// TIA Portal project "time_series_GV" (V14)

(* hardware
DEVICE "S71500/ET200MP station_1"  S7-1500 station
   slot 0: "Rail_0"  Rack  6ES7 590-1***0-0AA0
   slot 0: "PM 70W 120/230VAC"  PM 70W 120/230VAC  6EP1332-4BA00
   slot 1: "PLC_1"  CPU 1511-1 PN  6ES7 511-1AK01-0AB0  V2.1
      slot 3: "CPU display_1"  6ES7591-1AA00-0AA0
   slot 2: "DI 16/DQ 16x24VDC/0.5A BA_1"  DI 16/DQ 16x24VDC/0.5A BA  6ES7 523-1BL00-0AA0  V1.0
   slot 3: "AI/AQ 4xU/I/RTD/TC / 2xU/I ST_1"  AI/AQ 4xU/I/RTD/TC / 2xU/I ST  6ES7 534-7QE00-0AB0  V1.0
DEVICE "HMI_1"  KTP900 Basic PN
   slot 0: "KTP900 Basic PN"  KTP900 Basic PN  6AV2 123-2JB03-0AX0  14.0.1.0
   slot 1: "HMI_RT_1"  KTP900 Basic PN  6AV2 123-2JB03-0AX0  14.0.1.0
   slot 5: "HMI_1.IE_CP_1"  PROFINET Interface  14.0.1.0
      slot 1: "PROFINET Interface_1"  PROFINET Interface
         slot 1: "Port_1"  Port
*)

// ===== PLC "PLC_1"  CPU 1511-1 PN =====

VAR_GLOBAL   // PLC tag table "Default tag table"
   "System_Byte" AT %MB1 : Byte;
   "FirstScan" AT %M1.0 : Bool;
   "DiagStatusUpdate" AT %M1.1 : Bool;
   "AlwaysTRUE" AT %M1.2 : Bool;
   "AlwaysFALSE" AT %M1.3 : Bool;
   "Clock_Byte" AT %MB0 : Byte;
   "Clock_10Hz" AT %M0.0 : Bool;
   "Clock_5Hz" AT %M0.1 : Bool;
   "Clock_2.5Hz" AT %M0.2 : Bool;
   "Clock_2Hz" AT %M0.3 : Bool;
   "Clock_1.25Hz" AT %M0.4 : Bool;
   "Clock_1Hz" AT %M0.5 : Bool;
   "Clock_0.625Hz" AT %M0.6 : Bool;
   "Clock_0.5Hz" AT %M0.7 : Bool;
   "Out_Standart_Deviation" AT %MD2 : Real;
   "Cloc_frequence" AT %M6.0 : Bool;
   "countdown_Frequency" AT %MD8 : Time;
   "arithmetic_avg" AT %MD12 : Real;
   "stdt_out" AT %MD16 : Real;
   "error_avg" AT %M6.1 : Bool;
   "status_id" AT %MW20 : UInt;
   "status_bloc" AT %MW22 : Word;
   "ret_val_DB" AT %MW28 : Int;
   "value_read_array" AT %MW24 : Int;
   "ret_val_DB_read" AT %MW26 : Int;
   "size_array_block" AT %MW30 : Int;
   "signal_out_analog" AT %MW32 : Int;
   "standartDeviation" AT %MD34 : Real;
END_VAR

DATA_BLOCK "DB_Signal_measurement"   // DB1
{ S7_Optimized_Access := 'TRUE' }
VERSION : 0.1
   VAR
      Signal : Array[0..15] of Int;
   END_VAR
BEGIN
   Signal[0] := 1;
   Signal[1] := 2;
   Signal[2] := 3;
   Signal[4] := 5;
   Signal[3] := 4;
   Signal[5] := 6;
   Signal[6] := 7;
   Signal[7] := 8;
   Signal[8] := 9;
   Signal[9] := 0;
   Signal[10] := 1;
   Signal[11] := 2;
   Signal[12] := 3;
   Signal[13] := 4;
   Signal[14] := 5;
   Signal[15] := 6;
END_DATA_BLOCK

DATA_BLOCK "Array_DB_Signal"   // DB2
{ S7_Optimized_Access := 'TRUE' }
VERSION : 0.1
   VAR
      Header : ArrayDBHeader;
      THIS : Array[0..15] of Real;
   END_VAR
BEGIN
   Header.LowerBound := 0;
   Header.UpperBound := 15;
   Header.Elements := 16;
   Header.PaddedSize := 4;
   Header.ElementSize := 4;
   THIS[0] := 8.0;
   THIS[1] := 6.2;
   THIS[2] := 7.5;
   THIS[3] := 8.5;
   THIS[4] := 7.0;
   THIS[5] := 2.8;
   THIS[8] := 100.0;
   THIS[9] := 100.0;
END_DATA_BLOCK

DATA_BLOCK "HMI_Signal"   // DB3
{ S7_Optimized_Access := 'TRUE' }
VERSION : 0.1
   VAR
      HMI_signal_out_GV : Int;
      HMI_stdDeviation : Real;
   END_VAR
BEGIN
END_DATA_BLOCK

DATA_BLOCK "myArrayDB"   // DB4
{ S7_Optimized_Access := 'TRUE' }
VERSION : 0.1
   VAR
      Header : ArrayDBHeader;
      THIS : Array[0..1300] of Int;
   END_VAR
BEGIN
   Header.LowerBound := 0;
   Header.UpperBound := 1300;
   Header.Elements := 1301;
   Header.PaddedSize := 2;
   Header.ElementSize := 2;
   THIS[4] := 659;
   THIS[0] := 620;
   THIS[1] := 620;
   THIS[2] := 620;
   THIS[3] := 650;
   THIS[5] := 659;
   THIS[6] := 659;
   THIS[7] := 676;
   THIS[8] := 676;
   THIS[9] := 676;
   THIS[10] := 676;
   THIS[11] := 676;
   THIS[12] := 676;
   THIS[13] := 676;
   THIS[14] := 677;
   THIS[15] := 677;
   THIS[16] := 677;
   THIS[17] := 677;
   THIS[18] := 677;
   THIS[19] := 677;
   THIS[20] := 677;
   THIS[21] := 677;
   THIS[22] := 677;
   THIS[23] := 677;
   THIS[24] := 677;
   THIS[25] := 678;
   THIS[26] := 678;
   THIS[27] := 678;
   THIS[28] := 678;
   THIS[29] := 678;
   THIS[30] := 678;
   THIS[31] := 678;
   THIS[32] := 678;
   THIS[33] := 678;
   THIS[34] := 678;
   THIS[35] := 678;
   THIS[36] := 678;
   THIS[37] := 678;
   THIS[38] := 678;
   THIS[39] := 678;
   THIS[40] := 678;
   THIS[41] := 678;
   THIS[42] := 672;
   THIS[43] := 663;
   THIS[44] := 663;
   THIS[45] := 663;
   THIS[46] := 630;
   THIS[47] := 627;
   THIS[48] := 627;
   THIS[49] := 617;
   THIS[50] := 617;
   THIS[51] := 617;
   THIS[52] := 617;
   THIS[53] := 617;
   THIS[54] := 617;
   THIS[55] := 617;
   THIS[56] := 618;
   THIS[57] := 620;
   THIS[58] := 620;
   THIS[59] := 620;
   THIS[60] := 621;
   THIS[61] := 621;
   THIS[62] := 621;
   THIS[63] := 621;
   THIS[64] := 621;
   THIS[65] := 621;
   THIS[66] := 621;
   THIS[67] := 621;
   THIS[68] := 621;
   THIS[69] := 621;
   THIS[70] := 621;
   THIS[71] := 621;
   THIS[72] := 621;
   THIS[73] := 621;
   THIS[74] := 621;
   THIS[75] := 621;
   THIS[76] := 621;
   THIS[77] := 621;
   THIS[78] := 621;
   THIS[79] := 621;
   THIS[80] := 621;
   THIS[81] := 618;
   THIS[82] := 612;
   THIS[83] := 612;
   THIS[84] := 595;
   THIS[85] := 584;
   THIS[86] := 584;
   THIS[87] := 579;
   THIS[88] := 579;
   THIS[89] := 579;
   THIS[90] := 579;
   THIS[91] := 579;
   THIS[92] := 579;
   THIS[93] := 579;
   THIS[94] := 579;
   THIS[95] := 579;
   THIS[96] := 579;
   THIS[97] := 579;
   THIS[98] := 579;
   THIS[99] := 579;
   THIS[100] := 579;
   THIS[101] := 579;
   THIS[102] := 579;
   THIS[103] := 579;
   THIS[104] := 579;
   THIS[105] := 579;
   THIS[106] := 579;
   THIS[107] := 579;
   THIS[108] := 579;
   THIS[109] := 579;
   THIS[110] := 579;
   THIS[111] := 579;
   THIS[112] := 579;
   THIS[113] := 579;
   THIS[114] := 579;
   THIS[115] := 579;
   THIS[116] := 579;
   THIS[117] := 579;
   THIS[118] := 579;
   THIS[119] := 579;
   THIS[120] := 579;
   THIS[121] := 579;
   THIS[122] := 579;
   THIS[123] := 572;
   THIS[124] := 564;
   THIS[125] := 564;
   THIS[126] := 551;
   THIS[127] := 548;
   THIS[128] := 548;
   THIS[129] := 548;
   THIS[130] := 545;
   THIS[131] := 545;
   THIS[132] := 541;
   THIS[133] := 541;
   THIS[134] := 541;
   THIS[135] := 541;
   THIS[136] := 541;
   THIS[137] := 542;
   THIS[138] := 542;
   THIS[139] := 542;
   THIS[140] := 542;
   THIS[141] := 542;
   THIS[142] := 542;
   THIS[143] := 542;
   THIS[144] := 542;
   THIS[145] := 542;
   THIS[146] := 542;
   THIS[147] := 542;
   THIS[148] := 542;
   THIS[149] := 542;
   THIS[150] := 538;
   THIS[151] := 532;
   THIS[152] := 532;
   THIS[153] := 518;
   THIS[154] := 511;
   THIS[155] := 511;
   THIS[156] := 511;
   THIS[157] := 508;
   THIS[158] := 508;
   THIS[159] := 508;
   THIS[160] := 508;
   THIS[161] := 508;
   THIS[162] := 508;
   THIS[163] := 508;
   THIS[164] := 508;
   THIS[165] := 508;
   THIS[166] := 508;
   THIS[167] := 508;
   THIS[168] := 508;
   THIS[169] := 501;
   THIS[170] := 500;
   THIS[171] := 500;
   THIS[172] := 500;
   THIS[173] := 500;
   THIS[174] := 500;
   THIS[175] := 500;
   THIS[176] := 500;
   THIS[177] := 500;
   THIS[178] := 520;
   THIS[179] := 521;
   THIS[180] := 521;
   THIS[181] := 420;
   THIS[182] := 500;
   THIS[183] := 500;
   THIS[184] := 500;
   THIS[185] := 500;
   THIS[186] := 500;
   THIS[187] := 500;
   THIS[188] := 500;
   THIS[189] := 500;
   THIS[190] := 481;
   THIS[191] := 481;
   THIS[192] := 481;
   THIS[193] := 463;
   THIS[194] := 463;
   THIS[195] := 463;
   THIS[196] := 461;
   THIS[197] := 461;
   THIS[198] := 461;
   THIS[199] := 461;
   THIS[200] := 461;
   THIS[201] := 461;
   THIS[202] := 461;
   THIS[203] := 461;
   THIS[204] := 461;
   THIS[205] := 461;
   THIS[206] := 461;
   THIS[207] := 461;
   THIS[208] := 461;
   THIS[209] := 461;
   THIS[210] := 461;
   THIS[211] := 461;
   THIS[212] := 459;
   THIS[213] := 458;
   THIS[214] := 447;
   THIS[215] := 441;
   THIS[216] := 434;
   THIS[217] := 427;
   THIS[218] := 426;
   THIS[219] := 426;
   THIS[220] := 426;
   THIS[221] := 426;
   THIS[222] := 426;
   THIS[223] := 426;
   THIS[224] := 426;
   THIS[225] := 426;
   THIS[226] := 426;
   THIS[227] := 426;
   THIS[228] := 426;
   THIS[229] := 426;
   THIS[230] := 426;
   THIS[231] := 426;
   THIS[232] := 426;
   THIS[233] := 426;
   THIS[234] := 426;
   THIS[235] := 426;
   THIS[236] := 426;
   THIS[237] := 426;
   THIS[238] := 426;
   THIS[239] := 426;
   THIS[240] := 426;
   THIS[241] := 426;
   THIS[242] := 426;
   THIS[243] := 426;
   THIS[244] := 426;
   THIS[245] := 426;
   THIS[246] := 426;
   THIS[247] := 426;
   THIS[248] := 426;
   THIS[249] := 426;
   THIS[250] := 426;
   THIS[251] := 426;
   THIS[252] := 426;
   THIS[253] := 426;
   THIS[254] := 426;
   THIS[255] := 426;
   THIS[256] := 426;
   THIS[257] := 426;
   THIS[258] := 421;
   THIS[259] := 415;
   THIS[260] := 415;
   THIS[261] := 401;
   THIS[262] := 398;
   THIS[263] := 392;
   THIS[264] := 392;
   THIS[265] := 389;
   THIS[266] := 389;
   THIS[267] := 389;
   THIS[268] := 389;
   THIS[269] := 385;
   THIS[270] := 384;
   THIS[271] := 384;
   THIS[272] := 384;
   THIS[273] := 384;
   THIS[274] := 384;
   THIS[275] := 384;
   THIS[276] := 384;
   THIS[277] := 384;
   THIS[278] := 384;
   THIS[279] := 384;
   THIS[280] := 384;
   THIS[281] := 384;
   THIS[282] := 384;
   THIS[283] := 384;
   THIS[284] := 382;
   THIS[285] := 378;
   THIS[286] := 360;
   THIS[287] := 352;
   THIS[288] := 349;
   THIS[289] := 349;
   THIS[290] := 342;
   THIS[291] := 342;
   THIS[292] := 342;
   THIS[293] := 342;
   THIS[294] := 342;
   THIS[295] := 342;
   THIS[296] := 342;
   THIS[297] := 342;
   THIS[298] := 342;
   THIS[299] := 342;
   THIS[300] := 342;
   THIS[301] := 342;
   THIS[302] := 342;
   THIS[303] := 342;
   THIS[304] := 342;
   THIS[305] := 342;
   THIS[306] := 342;
   THIS[307] := 342;
   THIS[308] := 342;
   THIS[309] := 342;
   THIS[310] := 342;
   THIS[311] := 342;
   THIS[312] := 342;
   THIS[313] := 342;
   THIS[314] := 342;
   THIS[315] := 342;
   THIS[316] := 342;
   THIS[317] := 342;
   THIS[318] := 342;
   THIS[319] := 342;
   THIS[320] := 342;
   THIS[321] := 342;
   THIS[322] := 342;
   THIS[323] := 342;
   THIS[324] := 342;
   THIS[325] := 342;
   THIS[326] := 342;
   THIS[327] := 342;
   THIS[328] := 334;
   THIS[329] := 331;
   THIS[330] := 331;
   THIS[331] := 314;
   THIS[332] := 308;
   THIS[333] := 304;
   THIS[334] := 302;
   THIS[335] := 302;
   THIS[336] := 302;
   THIS[337] := 302;
   THIS[338] := 302;
   THIS[339] := 302;
   THIS[340] := 302;
   THIS[341] := 302;
   THIS[342] := 302;
   THIS[343] := 302;
   THIS[344] := 302;
   THIS[345] := 302;
   THIS[346] := 302;
   THIS[347] := 302;
   THIS[348] := 302;
   THIS[349] := 302;
   THIS[350] := 302;
   THIS[351] := 302;
   THIS[352] := 302;
   THIS[353] := 302;
   THIS[354] := 302;
   THIS[355] := 302;
   THIS[356] := 302;
   THIS[357] := 302;
   THIS[358] := 302;
   THIS[359] := 302;
   THIS[360] := 302;
   THIS[361] := 302;
   THIS[362] := 302;
   THIS[363] := 301;
   THIS[364] := 299;
   THIS[365] := 290;
   THIS[366] := 283;
   THIS[367] := 276;
   THIS[368] := 262;
   THIS[369] := 261;
   THIS[370] := 259;
   THIS[371] := 259;
   THIS[372] := 259;
   THIS[373] := 259;
   THIS[374] := 259;
   THIS[375] := 259;
   THIS[376] := 259;
   THIS[377] := 259;
   THIS[378] := 259;
   THIS[379] := 259;
   THIS[380] := 259;
   THIS[381] := 259;
   THIS[382] := 259;
   THIS[383] := 259;
   THIS[384] := 259;
   THIS[385] := 259;
   THIS[386] := 259;
   THIS[387] := 259;
   THIS[388] := 259;
   THIS[389] := 259;
   THIS[390] := 259;
   THIS[391] := 259;
   THIS[392] := 259;
   THIS[393] := 259;
   THIS[394] := 259;
   THIS[395] := 259;
   THIS[396] := 259;
   THIS[397] := 259;
   THIS[398] := 259;
   THIS[399] := 259;
   THIS[400] := 259;
   THIS[401] := 259;
   THIS[402] := 259;
   THIS[403] := 257;
   THIS[404] := 254;
   THIS[405] := 252;
   THIS[406] := 252;
   THIS[407] := 234;
   THIS[408] := 228;
   THIS[409] := 228;
   THIS[410] := 220;
   THIS[411] := 220;
   THIS[412] := 219;
   THIS[413] := 219;
   THIS[414] := 220;
   THIS[415] := 220;
   THIS[416] := 220;
   THIS[417] := 220;
   THIS[418] := 220;
   THIS[419] := 220;
   THIS[420] := 220;
   THIS[421] := 220;
   THIS[422] := 220;
   THIS[423] := 220;
   THIS[424] := 220;
   THIS[425] := 220;
   THIS[426] := 220;
   THIS[427] := 220;
   THIS[428] := 220;
   THIS[429] := 220;
   THIS[430] := 220;
   THIS[431] := 220;
   THIS[432] := 220;
   THIS[433] := 220;
   THIS[434] := 220;
   THIS[435] := 220;
   THIS[436] := 220;
   THIS[437] := 220;
   THIS[438] := 220;
   THIS[439] := 220;
   THIS[440] := 220;
   THIS[441] := 220;
   THIS[442] := 217;
   THIS[443] := 213;
   THIS[444] := 209;
   THIS[445] := 190;
   THIS[446] := 184;
   THIS[447] := 184;
   THIS[448] := 177;
   THIS[449] := 177;
   THIS[450] := 177;
   THIS[451] := 177;
   THIS[452] := 177;
   THIS[453] := 177;
   THIS[454] := 177;
   THIS[455] := 177;
   THIS[456] := 177;
   THIS[457] := 177;
   THIS[458] := 177;
   THIS[459] := 177;
   THIS[460] := 177;
   THIS[461] := 177;
   THIS[462] := 177;
   THIS[463] := 177;
   THIS[464] := 177;
   THIS[465] := 177;
   THIS[466] := 177;
   THIS[467] := 177;
   THIS[468] := 177;
   THIS[469] := 177;
   THIS[470] := 177;
   THIS[471] := 177;
   THIS[472] := 177;
   THIS[473] := 177;
   THIS[474] := 177;
   THIS[475] := 177;
   THIS[476] := 177;
   THIS[477] := 177;
   THIS[478] := 177;
   THIS[479] := 177;
   THIS[480] := 177;
   THIS[481] := 177;
   THIS[482] := 177;
   THIS[483] := 177;
   THIS[484] := 177;
   THIS[485] := 175;
   THIS[486] := 172;
   THIS[487] := 172;
   THIS[488] := 154;
   THIS[489] := 149;
   THIS[490] := 147;
   THIS[491] := 144;
   THIS[492] := 144;
   THIS[493] := 143;
   THIS[494] := 143;
   THIS[495] := 139;
   THIS[496] := 139;
   THIS[497] := 139;
   THIS[498] := 138;
   THIS[499] := 138;
   THIS[500] := 138;
   THIS[501] := 138;
   THIS[502] := 138;
   THIS[503] := 138;
   THIS[504] := 138;
   THIS[505] := 138;
   THIS[506] := 139;
   THIS[507] := 139;
   THIS[508] := 139;
   THIS[509] := 139;
   THIS[510] := 139;
   THIS[511] := 139;
   THIS[512] := 139;
   THIS[513] := 139;
   THIS[514] := 139;
   THIS[515] := 139;
   THIS[516] := 139;
   THIS[517] := 139;
   THIS[518] := 139;
   THIS[519] := 139;
   THIS[520] := 139;
   THIS[521] := 139;
   THIS[522] := 139;
   THIS[523] := 139;
   THIS[524] := 139;
   THIS[525] := 139;
   THIS[526] := 139;
   THIS[527] := 139;
   THIS[528] := 139;
   THIS[529] := 139;
   THIS[530] := 139;
   THIS[531] := 139;
   THIS[532] := 139;
   THIS[533] := 139;
   THIS[534] := 139;
   THIS[535] := 139;
   THIS[536] := 139;
   THIS[537] := 139;
   THIS[538] := 139;
   THIS[539] := 139;
   THIS[540] := 139;
   THIS[541] := 139;
   THIS[542] := 139;
   THIS[543] := 139;
   THIS[544] := 139;
   THIS[545] := 139;
   THIS[546] := 141;
   THIS[547] := 141;
   THIS[548] := 141;
   THIS[549] := 143;
   THIS[550] := 143;
   THIS[551] := 143;
   THIS[552] := 143;
   THIS[553] := 144;
   THIS[554] := 144;
   THIS[555] := 144;
   THIS[556] := 144;
   THIS[557] := 144;
   THIS[558] := 144;
   THIS[559] := 144;
   THIS[560] := 144;
   THIS[561] := 144;
   THIS[562] := 144;
   THIS[563] := 144;
   THIS[564] := 144;
   THIS[565] := 144;
   THIS[566] := 144;
   THIS[567] := 144;
   THIS[568] := 144;
   THIS[569] := 144;
   THIS[570] := 144;
   THIS[571] := 144;
   THIS[572] := 144;
   THIS[573] := 144;
   THIS[574] := 144;
   THIS[575] := 144;
   THIS[576] := 144;
   THIS[577] := 144;
   THIS[578] := 144;
   THIS[579] := 144;
   THIS[580] := 144;
   THIS[581] := 144;
   THIS[582] := 144;
   THIS[583] := 144;
   THIS[584] := 144;
   THIS[585] := 144;
   THIS[586] := 144;
   THIS[587] := 144;
   THIS[588] := 144;
   THIS[589] := 144;
   THIS[590] := 144;
   THIS[591] := 144;
   THIS[592] := 144;
   THIS[593] := 144;
   THIS[594] := 144;
   THIS[595] := 144;
   THIS[596] := 144;
   THIS[597] := 144;
   THIS[598] := 144;
   THIS[599] := 144;
   THIS[600] := 144;
   THIS[601] := 144;
   THIS[602] := 144;
   THIS[603] := 144;
   THIS[604] := 144;
   THIS[605] := 144;
   THIS[606] := 144;
   THIS[607] := 147;
   THIS[608] := 151;
   THIS[609] := 153;
   THIS[610] := 153;
   THIS[611] := 176;
   THIS[612] := 186;
   THIS[613] := 191;
   THIS[614] := 217;
   THIS[615] := 229;
   THIS[616] := 242;
   THIS[617] := 242;
   THIS[618] := 269;
   THIS[619] := 288;
   THIS[620] := 288;
   THIS[621] := 320;
   THIS[622] := 334;
   THIS[623] := 340;
   THIS[624] := 340;
   THIS[625] := 389;
   THIS[626] := 395;
   THIS[627] := 395;
   THIS[628] := 434;
   THIS[629] := 441;
   THIS[630] := 441;
   THIS[631] := 485;
   THIS[632] := 492;
   THIS[633] := 492;
   THIS[634] := 537;
   THIS[635] := 548;
   THIS[636] := 548;
   THIS[637] := 593;
   THIS[638] := 593;
   THIS[639] := 593;
   THIS[640] := 638;
   THIS[641] := 638;
   THIS[642] := 665;
   THIS[643] := 670;
   THIS[644] := 670;
   THIS[645] := 670;
   THIS[646] := 674;
   THIS[647] := 674;
   THIS[648] := 674;
   THIS[649] := 674;
   THIS[650] := 674;
   THIS[651] := 674;
   THIS[652] := 674;
   THIS[653] := 674;
   THIS[654] := 674;
   THIS[655] := 674;
   THIS[656] := 674;
   THIS[657] := 674;
   THIS[658] := 674;
   THIS[659] := 674;
   THIS[660] := 674;
   THIS[661] := 674;
   THIS[662] := 674;
   THIS[663] := 674;
   THIS[664] := 675;
   THIS[665] := 675;
   THIS[666] := 675;
   THIS[667] := 675;
   THIS[668] := 675;
   THIS[669] := 675;
   THIS[670] := 675;
   THIS[671] := 675;
   THIS[672] := 675;
   THIS[673] := 675;
   THIS[674] := 675;
   THIS[675] := 675;
   THIS[676] := 675;
   THIS[677] := 675;
   THIS[678] := 675;
   THIS[679] := 675;
   THIS[680] := 674;
   THIS[681] := 671;
   THIS[682] := 669;
   THIS[683] := 669;
   THIS[684] := 649;
   THIS[685] := 642;
   THIS[686] := 642;
   THIS[687] := 633;
   THIS[688] := 633;
   THIS[689] := 633;
   THIS[690] := 631;
   THIS[691] := 628;
   THIS[692] := 628;
   THIS[693] := 626;
   THIS[694] := 626;
   THIS[695] := 626;
   THIS[696] := 626;
   THIS[697] := 626;
   THIS[698] := 626;
   THIS[699] := 626;
   THIS[700] := 626;
   THIS[701] := 626;
   THIS[702] := 626;
   THIS[703] := 626;
   THIS[704] := 626;
   THIS[705] := 626;
   THIS[706] := 626;
   THIS[707] := 626;
   THIS[708] := 626;
   THIS[709] := 626;
   THIS[710] := 626;
   THIS[711] := 626;
   THIS[712] := 626;
   THIS[713] := 626;
   THIS[714] := 626;
   THIS[715] := 626;
   THIS[716] := 626;
   THIS[717] := 626;
   THIS[718] := 626;
   THIS[719] := 626;
   THIS[720] := 625;
   THIS[721] := 625;
   THIS[722] := 618;
   THIS[723] := 612;
   THIS[724] := 609;
   THIS[725] := 609;
   THIS[726] := 591;
   THIS[727] := 584;
   THIS[728] := 584;
   THIS[729] := 584;
   THIS[730] := 582;
   THIS[731] := 582;
   THIS[732] := 582;
   THIS[733] := 582;
   THIS[734] := 582;
   THIS[735] := 582;
   THIS[736] := 582;
   THIS[737] := 582;
   THIS[738] := 582;
   THIS[739] := 582;
   THIS[740] := 582;
   THIS[741] := 582;
   THIS[742] := 582;
   THIS[743] := 582;
   THIS[744] := 582;
   THIS[745] := 582;
   THIS[746] := 582;
   THIS[747] := 582;
   THIS[748] := 582;
   THIS[749] := 582;
   THIS[750] := 582;
   THIS[751] := 582;
   THIS[752] := 582;
   THIS[753] := 582;
   THIS[754] := 582;
   THIS[755] := 582;
   THIS[756] := 582;
   THIS[757] := 582;
   THIS[758] := 582;
   THIS[759] := 582;
   THIS[760] := 582;
   THIS[761] := 582;
   THIS[762] := 582;
   THIS[763] := 582;
   THIS[764] := 582;
   THIS[765] := 583;
   THIS[766] := 580;
   THIS[767] := 580;
   THIS[768] := 569;
   THIS[769] := 559;
   THIS[770] := 559;
   THIS[771] := 559;
   THIS[772] := 548;
   THIS[773] := 548;
   THIS[774] := 548;
   THIS[775] := 546;
   THIS[776] := 543;
   THIS[777] := 543;
   THIS[778] := 540;
   THIS[779] := 540;
   THIS[780] := 540;
   THIS[781] := 540;
   THIS[782] := 541;
   THIS[783] := 541;
   THIS[784] := 541;
   THIS[785] := 541;
   THIS[786] := 541;
   THIS[787] := 541;
   THIS[788] := 541;
   THIS[789] := 541;
   THIS[790] := 541;
   THIS[791] := 541;
   THIS[792] := 541;
   THIS[793] := 541;
   THIS[794] := 541;
   THIS[795] := 541;
   THIS[796] := 541;
   THIS[797] := 539;
   THIS[798] := 536;
   THIS[799] := 532;
   THIS[800] := 532;
   THIS[801] := 518;
   THIS[802] := 510;
   THIS[803] := 510;
   THIS[804] := 510;
   THIS[805] := 503;
   THIS[806] := 503;
   THIS[807] := 503;
   THIS[808] := 503;
   THIS[809] := 503;
   THIS[810] := 503;
   THIS[811] := 503;
   THIS[812] := 503;
   THIS[813] := 503;
   THIS[814] := 503;
   THIS[815] := 503;
   THIS[816] := 503;
   THIS[817] := 503;
   THIS[818] := 503;
   THIS[819] := 503;
   THIS[820] := 503;
   THIS[821] := 503;
   THIS[822] := 503;
   THIS[823] := 503;
   THIS[824] := 503;
   THIS[825] := 503;
   THIS[826] := 503;
   THIS[827] := 503;
   THIS[828] := 503;
   THIS[829] := 503;
   THIS[830] := 503;
   THIS[831] := 503;
   THIS[832] := 503;
   THIS[833] := 503;
   THIS[834] := 503;
   THIS[835] := 503;
   THIS[836] := 503;
   THIS[837] := 502;
   THIS[838] := 502;
   THIS[839] := 494;
   THIS[840] := 488;
   THIS[841] := 481;
   THIS[842] := 481;
   THIS[843] := 465;
   THIS[844] := 459;
   THIS[845] := 459;
   THIS[846] := 455;
   THIS[847] := 455;
   THIS[848] := 455;
   THIS[849] := 458;
   THIS[850] := 459;
   THIS[851] := 459;
   THIS[852] := 459;
   THIS[853] := 459;
   THIS[854] := 459;
   THIS[855] := 459;
   THIS[856] := 459;
   THIS[857] := 459;
   THIS[858] := 459;
   THIS[859] := 459;
   THIS[860] := 459;
   THIS[861] := 459;
   THIS[862] := 459;
   THIS[863] := 459;
   THIS[864] := 459;
   THIS[865] := 459;
   THIS[866] := 459;
   THIS[867] := 459;
   THIS[868] := 459;
   THIS[869] := 459;
   THIS[870] := 448;
   THIS[871] := 438;
   THIS[872] := 438;
   THIS[873] := 422;
   THIS[874] := 419;
   THIS[875] := 419;
   THIS[876] := 419;
   THIS[877] := 419;
   THIS[878] := 419;
   THIS[879] := 419;
   THIS[880] := 419;
   THIS[881] := 419;
   THIS[882] := 419;
   THIS[883] := 419;
   THIS[884] := 419;
   THIS[885] := 419;
   THIS[886] := 419;
   THIS[887] := 419;
   THIS[888] := 419;
   THIS[889] := 419;
   THIS[890] := 419;
   THIS[891] := 419;
   THIS[892] := 419;
   THIS[893] := 419;
   THIS[894] := 419;
   THIS[895] := 419;
   THIS[896] := 419;
   THIS[897] := 419;
   THIS[898] := 419;
   THIS[899] := 419;
   THIS[900] := 419;
   THIS[901] := 419;
   THIS[902] := 419;
   THIS[903] := 419;
   THIS[904] := 419;
   THIS[905] := 419;
   THIS[906] := 418;
   THIS[907] := 418;
   THIS[908] := 408;
   THIS[909] := 402;
   THIS[910] := 399;
   THIS[911] := 385;
   THIS[912] := 382;
   THIS[913] := 382;
   THIS[914] := 382;
   THIS[915] := 381;
   THIS[916] := 381;
   THIS[917] := 381;
   THIS[918] := 381;
   THIS[919] := 381;
   THIS[920] := 381;
   THIS[921] := 381;
   THIS[922] := 381;
   THIS[923] := 381;
   THIS[924] := 381;
   THIS[925] := 381;
   THIS[926] := 381;
   THIS[927] := 381;
   THIS[928] := 381;
   THIS[929] := 381;
   THIS[930] := 381;
   THIS[931] := 381;
   THIS[932] := 381;
   THIS[933] := 381;
   THIS[934] := 381;
   THIS[935] := 381;
   THIS[936] := 381;
   THIS[937] := 379;
   THIS[938] := 379;
   THIS[939] := 371;
   THIS[940] := 359;
   THIS[941] := 359;
   THIS[942] := 359;
   THIS[943] := 341;
   THIS[944] := 340;
   THIS[945] := 340;
   THIS[946] := 339;
   THIS[947] := 339;
   THIS[948] := 339;
   THIS[949] := 339;
   THIS[950] := 339;
   THIS[951] := 339;
   THIS[952] := 339;
   THIS[953] := 339;
   THIS[954] := 339;
   THIS[955] := 339;
   THIS[956] := 339;
   THIS[957] := 339;
   THIS[958] := 339;
   THIS[959] := 339;
   THIS[960] := 339;
   THIS[961] := 339;
   THIS[962] := 339;
   THIS[963] := 339;
   THIS[964] := 339;
   THIS[965] := 339;
   THIS[966] := 339;
   THIS[967] := 339;
   THIS[968] := 339;
   THIS[969] := 339;
   THIS[970] := 339;
   THIS[971] := 339;
   THIS[972] := 339;
   THIS[973] := 339;
   THIS[974] := 339;
   THIS[975] := 339;
   THIS[976] := 339;
   THIS[977] := 339;
   THIS[978] := 339;
   THIS[979] := 339;
   THIS[980] := 339;
   THIS[981] := 339;
   THIS[982] := 339;
   THIS[983] := 339;
   THIS[984] := 332;
   THIS[985] := 324;
   THIS[986] := 324;
   THIS[987] := 324;
   THIS[988] := 300;
   THIS[989] := 298;
   THIS[990] := 298;
   THIS[991] := 296;
   THIS[992] := 296;
   THIS[993] := 296;
   THIS[994] := 296;
   THIS[995] := 296;
   THIS[996] := 296;
   THIS[997] := 296;
   THIS[998] := 296;
   THIS[999] := 296;
   THIS[1000] := 296;
   THIS[1001] := 296;
   THIS[1002] := 296;
   THIS[1003] := 296;
   THIS[1004] := 296;
   THIS[1005] := 296;
   THIS[1006] := 296;
   THIS[1007] := 296;
   THIS[1008] := 296;
   THIS[1009] := 296;
   THIS[1010] := 296;
   THIS[1011] := 296;
   THIS[1012] := 296;
   THIS[1013] := 296;
   THIS[1014] := 295;
   THIS[1015] := 291;
   THIS[1016] := 291;
   THIS[1017] := 291;
   THIS[1018] := 268;
   THIS[1019] := 264;
   THIS[1020] := 264;
   THIS[1021] := 252;
   THIS[1022] := 252;
   THIS[1023] := 252;
   THIS[1024] := 252;
   THIS[1025] := 252;
   THIS[1026] := 252;
   THIS[1027] := 252;
   THIS[1028] := 252;
   THIS[1029] := 252;
   THIS[1030] := 252;
   THIS[1031] := 252;
   THIS[1032] := 252;
   THIS[1033] := 252;
   THIS[1034] := 252;
   THIS[1035] := 252;
   THIS[1036] := 252;
   THIS[1037] := 252;
   THIS[1038] := 252;
   THIS[1039] := 252;
   THIS[1040] := 252;
   THIS[1041] := 252;
   THIS[1042] := 252;
   THIS[1043] := 252;
   THIS[1044] := 252;
   THIS[1045] := 252;
   THIS[1046] := 252;
   THIS[1047] := 252;
   THIS[1048] := 252;
   THIS[1049] := 252;
   THIS[1050] := 252;
   THIS[1051] := 252;
   THIS[1052] := 252;
   THIS[1053] := 252;
   THIS[1054] := 252;
   THIS[1055] := 252;
   THIS[1056] := 252;
   THIS[1057] := 252;
   THIS[1058] := 252;
   THIS[1059] := 252;
   THIS[1060] := 252;
   THIS[1061] := 252;
   THIS[1062] := 252;
   THIS[1063] := 245;
   THIS[1064] := 243;
   THIS[1065] := 243;
   THIS[1066] := 224;
   THIS[1067] := 219;
   THIS[1068] := 219;
   THIS[1069] := 217;
   THIS[1070] := 217;
   THIS[1071] := 217;
   THIS[1072] := 217;
   THIS[1073] := 217;
   THIS[1074] := 217;
   THIS[1075] := 217;
   THIS[1076] := 217;
   THIS[1077] := 217;
   THIS[1078] := 217;
   THIS[1079] := 217;
   THIS[1080] := 217;
   THIS[1081] := 217;
   THIS[1082] := 217;
   THIS[1083] := 217;
   THIS[1084] := 217;
   THIS[1085] := 217;
   THIS[1086] := 217;
   THIS[1087] := 217;
   THIS[1088] := 217;
   THIS[1089] := 217;
   THIS[1090] := 217;
   THIS[1091] := 217;
   THIS[1092] := 217;
   THIS[1093] := 217;
   THIS[1094] := 217;
   THIS[1095] := 217;
   THIS[1096] := 217;
   THIS[1097] := 217;
   THIS[1098] := 217;
   THIS[1099] := 217;
   THIS[1100] := 217;
   THIS[1101] := 217;
   THIS[1102] := 215;
   THIS[1103] := 215;
   THIS[1104] := 204;
   THIS[1105] := 197;
   THIS[1106] := 182;
   THIS[1107] := 179;
   THIS[1108] := 179;
   THIS[1109] := 179;
   THIS[1110] := 179;
   THIS[1111] := 179;
   THIS[1112] := 179;
   THIS[1113] := 179;
   THIS[1114] := 179;
   THIS[1115] := 179;
   THIS[1116] := 179;
   THIS[1117] := 179;
   THIS[1118] := 179;
   THIS[1119] := 179;
   THIS[1120] := 179;
   THIS[1121] := 179;
   THIS[1122] := 179;
   THIS[1123] := 179;
   THIS[1124] := 179;
   THIS[1125] := 179;
   THIS[1126] := 179;
   THIS[1127] := 179;
   THIS[1128] := 179;
   THIS[1129] := 179;
   THIS[1130] := 179;
   THIS[1131] := 179;
   THIS[1132] := 179;
   THIS[1133] := 179;
   THIS[1134] := 179;
   THIS[1135] := 179;
   THIS[1136] := 179;
   THIS[1137] := 179;
   THIS[1138] := 179;
   THIS[1139] := 179;
   THIS[1140] := 179;
   THIS[1141] := 179;
   THIS[1142] := 179;
   THIS[1143] := 179;
   THIS[1144] := 179;
   THIS[1145] := 179;
   THIS[1146] := 179;
   THIS[1147] := 164;
   THIS[1148] := 164;
   THIS[1149] := 164;
   THIS[1150] := 148;
   THIS[1151] := 148;
   THIS[1152] := 148;
   THIS[1153] := 148;
   THIS[1154] := 148;
   THIS[1155] := 148;
   THIS[1156] := 141;
   THIS[1157] := 141;
   THIS[1158] := 141;
   THIS[1159] := 141;
   THIS[1160] := 141;
   THIS[1161] := 141;
   THIS[1162] := 139;
   THIS[1163] := 139;
   THIS[1164] := 139;
   THIS[1165] := 139;
   THIS[1166] := 139;
   THIS[1167] := 139;
   THIS[1168] := 139;
   THIS[1169] := 139;
   THIS[1170] := 139;
   THIS[1171] := 139;
   THIS[1172] := 139;
   THIS[1173] := 139;
   THIS[1174] := 139;
   THIS[1175] := 139;
   THIS[1176] := 139;
   THIS[1177] := 139;
   THIS[1178] := 139;
   THIS[1179] := 139;
   THIS[1180] := 139;
   THIS[1181] := 139;
   THIS[1182] := 139;
   THIS[1183] := 139;
   THIS[1184] := 139;
   THIS[1185] := 139;
   THIS[1186] := 139;
   THIS[1187] := 139;
   THIS[1188] := 139;
   THIS[1189] := 139;
   THIS[1190] := 139;
   THIS[1191] := 139;
   THIS[1192] := 139;
   THIS[1193] := 139;
   THIS[1194] := 139;
   THIS[1195] := 139;
   THIS[1196] := 139;
   THIS[1197] := 139;
   THIS[1198] := 140;
   THIS[1199] := 143;
   THIS[1200] := 144;
   THIS[1201] := 144;
   THIS[1202] := 144;
   THIS[1203] := 144;
   THIS[1204] := 144;
   THIS[1205] := 144;
   THIS[1206] := 144;
   THIS[1207] := 144;
   THIS[1208] := 144;
   THIS[1209] := 144;
   THIS[1210] := 144;
   THIS[1211] := 144;
   THIS[1212] := 144;
   THIS[1213] := 144;
   THIS[1214] := 144;
   THIS[1215] := 144;
   THIS[1216] := 144;
   THIS[1217] := 144;
   THIS[1218] := 144;
   THIS[1219] := 144;
   THIS[1220] := 144;
   THIS[1221] := 144;
   THIS[1222] := 144;
   THIS[1223] := 144;
   THIS[1224] := 144;
   THIS[1225] := 144;
   THIS[1226] := 144;
   THIS[1227] := 144;
   THIS[1228] := 144;
   THIS[1229] := 144;
   THIS[1230] := 144;
   THIS[1231] := 144;
   THIS[1232] := 144;
   THIS[1233] := 144;
   THIS[1234] := 144;
   THIS[1235] := 144;
   THIS[1236] := 144;
   THIS[1237] := 144;
   THIS[1238] := 144;
   THIS[1239] := 144;
   THIS[1240] := 144;
   THIS[1241] := 144;
   THIS[1242] := 144;
   THIS[1243] := 144;
   THIS[1244] := 144;
   THIS[1245] := 144;
   THIS[1246] := 144;
   THIS[1247] := 144;
   THIS[1248] := 144;
   THIS[1249] := 144;
   THIS[1250] := 144;
   THIS[1251] := 144;
   THIS[1252] := 144;
   THIS[1253] := 144;
   THIS[1254] := 144;
   THIS[1255] := 146;
   THIS[1256] := 146;
   THIS[1257] := 161;
   THIS[1258] := 179;
   THIS[1259] := 179;
   THIS[1260] := 209;
   THIS[1261] := 227;
   THIS[1262] := 227;
   THIS[1263] := 227;
   THIS[1264] := 273;
   THIS[1265] := 278;
   THIS[1266] := 278;
   THIS[1267] := 317;
   THIS[1268] := 323;
   THIS[1269] := 323;
   THIS[1270] := 363;
   THIS[1271] := 376;
   THIS[1272] := 376;
   THIS[1273] := 407;
   THIS[1274] := 421;
   THIS[1275] := 427;
   THIS[1276] := 427;
   THIS[1277] := 464;
   THIS[1278] := 476;
   THIS[1279] := 482;
   THIS[1280] := 509;
   THIS[1281] := 522;
   THIS[1282] := 528;
   THIS[1283] := 528;
   THIS[1284] := 567;
   THIS[1285] := 579;
   THIS[1286] := 579;
   THIS[1287] := 611;
   THIS[1288] := 629;
   THIS[1289] := 636;
   THIS[1290] := 636;
   THIS[1291] := 663;
   THIS[1292] := 663;
   THIS[1293] := 663;
   THIS[1294] := 671;
   THIS[1295] := 671;
   THIS[1296] := 671;
   THIS[1297] := 671;
   THIS[1298] := 672;
   THIS[1299] := 672;
   THIS[1300] := 673;
END_DATA_BLOCK

DATA_BLOCK "AlarmHMI_DB"   // DB5
{ S7_Optimized_Access := 'TRUE' }
VERSION : 0.1
   VAR
      bAlarm_bool : Array[0..15] of Bool;
      wAlarm : Word;
   END_VAR
BEGIN
END_DATA_BLOCK

DATA_BLOCK "Signal_To_array_DB"   // DB9
{ S7_Optimized_Access := 'TRUE' }
VERSION : 0.1
   VAR
      Header : ArrayDBHeader;
      THIS : Array[0..5] of Int;
   END_VAR
BEGIN
   Header.LowerBound := 0;
   Header.UpperBound := 5;
   Header.Elements := 6;
   Header.PaddedSize := 2;
   Header.ElementSize := 2;
END_DATA_BLOCK

DATA_BLOCK "Alarm_FB_DB"   // DB11
{ S7_Optimized_Access := 'TRUE' }
VERSION : 0.1
// stored: InstanceOfName Alarm_FB
"Alarm_FB"
BEGIN
END_DATA_BLOCK

// folder: System blocks/Program resources

DATA_BLOCK "counter_ctu"   // DB6
{ S7_Optimized_Access := 'TRUE' }
AUTHOR : Simatic
FAMILY : IEC
NAME : CNTR
VERSION : 1.0
// stored: InstanceOfName IEC_COUNTER
"IEC_COUNTER"
BEGIN
END_DATA_BLOCK

DATA_BLOCK "ctu_blok_signal"   // DB7
{ S7_Optimized_Access := 'TRUE' }
AUTHOR : Simatic
FAMILY : IEC
NAME : CNTR
VERSION : 1.0
// stored: InstanceOfName IEC_COUNTER
"IEC_COUNTER"
BEGIN
END_DATA_BLOCK

DATA_BLOCK "IEC_Timer_0_DB"   // DB8
{ S7_Optimized_Access := 'TRUE' }
AUTHOR : Simatic
FAMILY : IEC
NAME : IEC_TMR
VERSION : 1.0
// stored: InstanceOfName IEC_TIMER
"IEC_TIMER"
BEGIN
END_DATA_BLOCK

DATA_BLOCK "IEC_Timer_0_DB_1"   // DB10
{ S7_Optimized_Access := 'TRUE' }
AUTHOR : Simatic
FAMILY : IEC
NAME : IEC_TMR
VERSION : 1.0
// stored: InstanceOfName IEC_TIMER
"IEC_TIMER"
BEGIN
END_DATA_BLOCK

// folder: (top level)

FUNCTION_BLOCK "Alarm_FB"   // FB1, LAD
{ S7_Optimized_Access := 'TRUE' }
VERSION : 0.1
   VAR_INPUT
      in1 : Bool;
      in2 : Bool;
      in3 : Bool;
      in4 : Bool;
      in5 : Bool;
      in6 : Bool;
      in7 : Bool;
      in8 : Bool;
      in9 : Bool;
      in10 : Bool;
      in11 : Bool;
      in12 : Bool;
      in13 : Bool;
      In14 : Bool;
      in15 : Bool;
      in16 : Bool;
   END_VAR
   VAR_OUTPUT
      ourWordAlarm : Word;
   END_VAR
   VAR
      alarm_word : Word;
      alarm_bool AT alarm_word : Array[0..15] of Bool;
   END_VAR
BEGIN

REGION Network 1
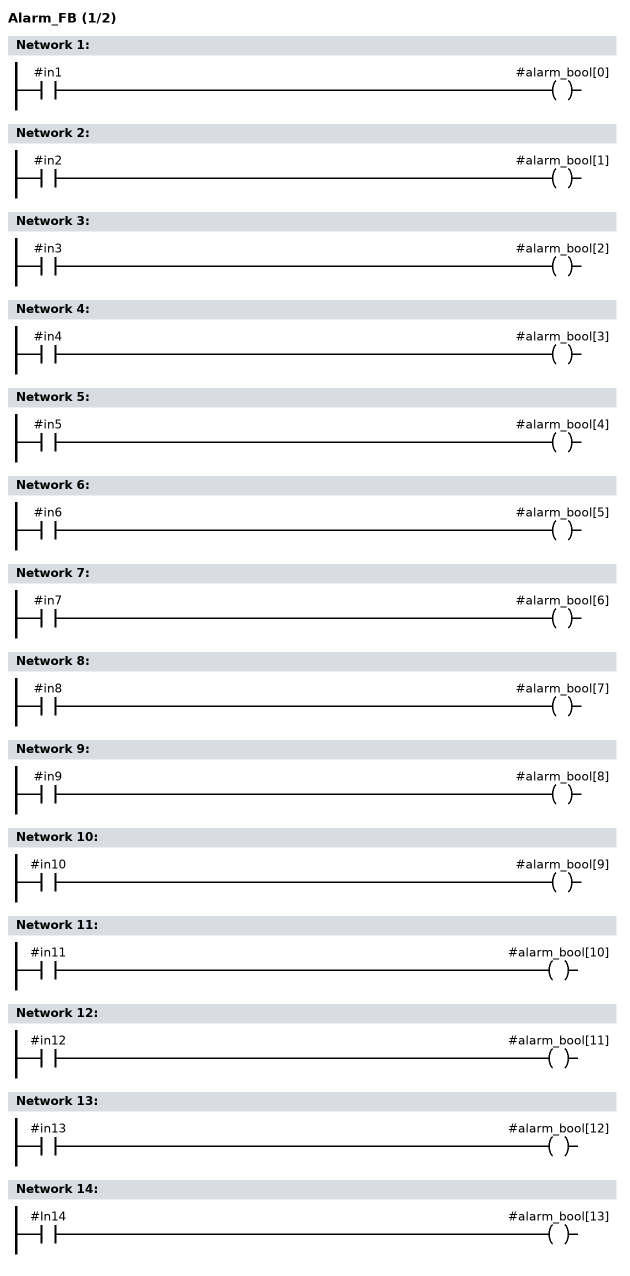
   RUNG wire#powerrail
      Contact( #in1 )
      Coil( #alarm_bool[0] )
   END_RUNG
   // the same network as SCL:
   #alarm_bool[0] := #in1;
END_REGION

REGION Network 2
   RUNG wire#powerrail
      Contact( #in2 )
      Coil( #alarm_bool[1] )
   END_RUNG
   // the same network as SCL:
   #alarm_bool[1] := #in2;
END_REGION

REGION Network 3
   RUNG wire#powerrail
      Contact( #in3 )
      Coil( #alarm_bool[2] )
   END_RUNG
   // the same network as SCL:
   #alarm_bool[2] := #in3;
END_REGION

REGION Network 4
   RUNG wire#powerrail
      Contact( #in4 )
      Coil( #alarm_bool[3] )
   END_RUNG
   // the same network as SCL:
   #alarm_bool[3] := #in4;
END_REGION

REGION Network 5
   RUNG wire#powerrail
      Contact( #in5 )
      Coil( #alarm_bool[4] )
   END_RUNG
   // the same network as SCL:
   #alarm_bool[4] := #in5;
END_REGION

REGION Network 6
   RUNG wire#powerrail
      Contact( #in6 )
      Coil( #alarm_bool[5] )
   END_RUNG
   // the same network as SCL:
   #alarm_bool[5] := #in6;
END_REGION

REGION Network 7
   RUNG wire#powerrail
      Contact( #in7 )
      Coil( #alarm_bool[6] )
   END_RUNG
   // the same network as SCL:
   #alarm_bool[6] := #in7;
END_REGION

REGION Network 8
   RUNG wire#powerrail
      Contact( #in8 )
      Coil( #alarm_bool[7] )
   END_RUNG
   // the same network as SCL:
   #alarm_bool[7] := #in8;
END_REGION

REGION Network 9
   RUNG wire#powerrail
      Contact( #in9 )
      Coil( #alarm_bool[8] )
   END_RUNG
   // the same network as SCL:
   #alarm_bool[8] := #in9;
END_REGION

REGION Network 10
   RUNG wire#powerrail
      Contact( #in10 )
      Coil( #alarm_bool[9] )
   END_RUNG
   // the same network as SCL:
   #alarm_bool[9] := #in10;
END_REGION

REGION Network 11
   RUNG wire#powerrail
      Contact( #in11 )
      Coil( #alarm_bool[10] )
   END_RUNG
   // the same network as SCL:
   #alarm_bool[10] := #in11;
END_REGION

REGION Network 12
   RUNG wire#powerrail
      Contact( #in12 )
      Coil( #alarm_bool[11] )
   END_RUNG
   // the same network as SCL:
   #alarm_bool[11] := #in12;
END_REGION

REGION Network 13
   RUNG wire#powerrail
      Contact( #in13 )
      Coil( #alarm_bool[12] )
   END_RUNG
   // the same network as SCL:
   #alarm_bool[12] := #in13;
END_REGION

REGION Network 14
   RUNG wire#powerrail
      Contact( #In14 )
      Coil( #alarm_bool[13] )
   END_RUNG
   // the same network as SCL:
   #alarm_bool[13] := #In14;
END_REGION

REGION Network 15
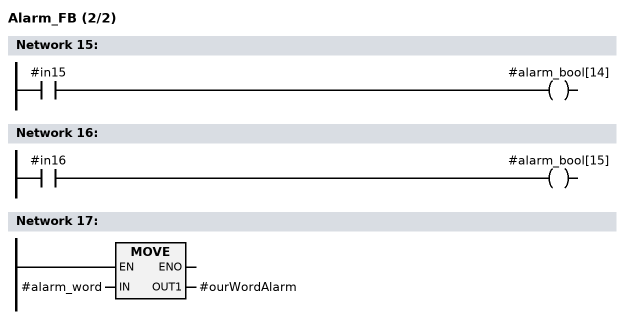
   RUNG wire#powerrail
      Contact( #in15 )
      Coil( #alarm_bool[14] )
   END_RUNG
   // the same network as SCL:
   #alarm_bool[14] := #in15;
END_REGION

REGION Network 16
   RUNG wire#powerrail
      Contact( #in16 )
      Coil( #alarm_bool[15] )
   END_RUNG
   // the same network as SCL:
   #alarm_bool[15] := #in16;
END_REGION

REGION Network 17
   RUNG wire#powerrail
      Move(in := #alarm_word, out1 => #ourWordAlarm)
   END_RUNG
   // the same network as SCL:
   #ourWordAlarm := #alarm_word;
END_REGION
END_FUNCTION_BLOCK

FUNCTION "signal_to_array_FC" : Void   // FC1, LAD
{ S7_Optimized_Access := 'TRUE' }
VERSION : 0.1
   VAR_INPUT
      signal : Int;
   END_VAR
   VAR_TEMP
      count : Bool;
      timer_freq : Time;
      memory : Bool;
      index : Int;
   END_VAR
BEGIN

REGION Network 1
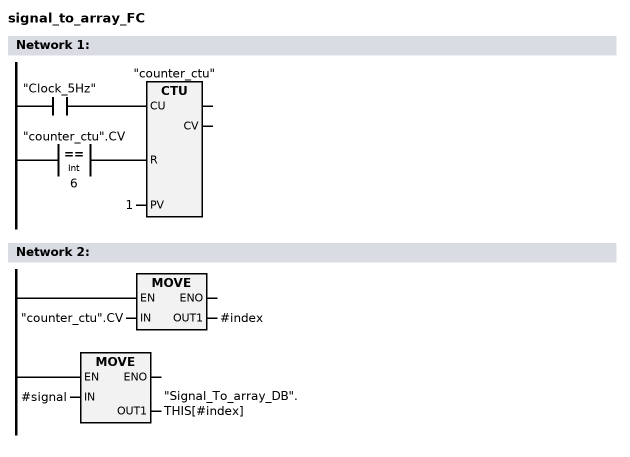
   "counter_ctu".CTU(CU := "Clock_5Hz", R := "counter_ctu".CV = 6, PV := 1);
END_REGION

REGION Network 2
   RUNG wire#powerrail
      Move(in := "counter_ctu".CV, out1 => #index)
   END_RUNG
   RUNG wire#powerrail
      Move(in := #signal, out1 => "Signal_To_array_DB".THIS[#index])
   END_RUNG
   // the same network as SCL:
   #index := "counter_ctu".CV;
   "Signal_To_array_DB".THIS[#index] := #signal;
END_REGION
END_FUNCTION

FUNCTION "Block_signal_modulator" : Void   // FC3, LAD
{ S7_Optimized_Access := 'TRUE' }
VERSION : 0.1
   VAR_INPUT
      variableArray : Variant;
      array_db : DB_ANY;
   END_VAR
   VAR_OUTPUT
      Signal_out : Int;
   END_VAR
   VAR_IN_OUT
      signal_HMI : Int;
   END_VAR
   VAR_TEMP
      tempArraySize : Int;
      reset_bloc_ctu : Bool;
      reset_ctu : Bool;
      ret_val_1 : Int;
      reset : Bool;
   END_VAR
BEGIN

REGION Network 1 (SCL)
   #tempArraySize := CountOfElements(#variableArray);
END_REGION

REGION Network 2 (SCL)
   IF "ctu_blok_signal".CV> #tempArraySize THEN
       #reset := TRUE;
   END_IF;
   "counter_ctu".R := #reset;
END_REGION

REGION Network 3
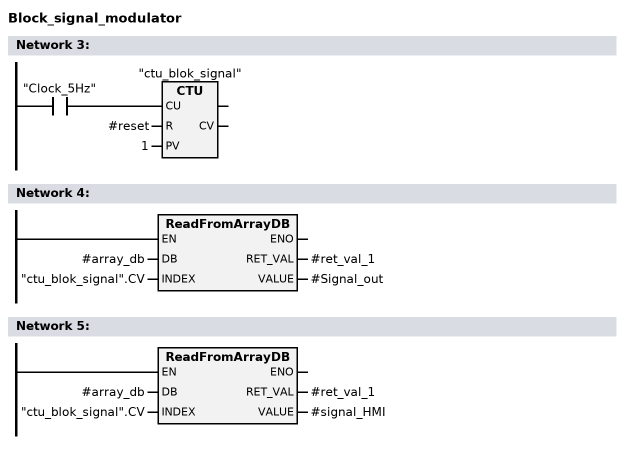
   "ctu_blok_signal".CTU(CU := "Clock_5Hz", R := #reset, PV := 1);
END_REGION

REGION Network 4
   // no SCL statement known for ReadFromArrayDB: written as a call
   #ret_val_1 := ReadFromArrayDB(db := #array_db, index := "ctu_blok_signal".CV, value => #Signal_out);
END_REGION

REGION Network 5
   // no SCL statement known for ReadFromArrayDB: written as a call
   #ret_val_1 := ReadFromArrayDB(db := #array_db, index := "ctu_blok_signal".CV, value => #signal_HMI);
END_REGION
END_FUNCTION

ORGANIZATION_BLOCK "Main"   // OB1, LAD, ProgramCycle
TITLE = "Main Program Sweep (Cycle)"
{ S7_Optimized_Access := 'TRUE' }
VERSION : 0.1
   VAR_INPUT
      Initial_Call : Bool;   // Initial call of this OB
      Remanence : Bool;   // =True, if remanent data are available
   END_VAR
   VAR_TEMP
      signal : Variant;
      ret_val_variant : Int;
      Aver : Real;
      Deviat : Real;
   END_VAR
   VAR_TEMP   // added for the SCL form of the ladder/FBD networks
      _w1 : Bool;
   END_VAR
BEGIN

REGION Network 1
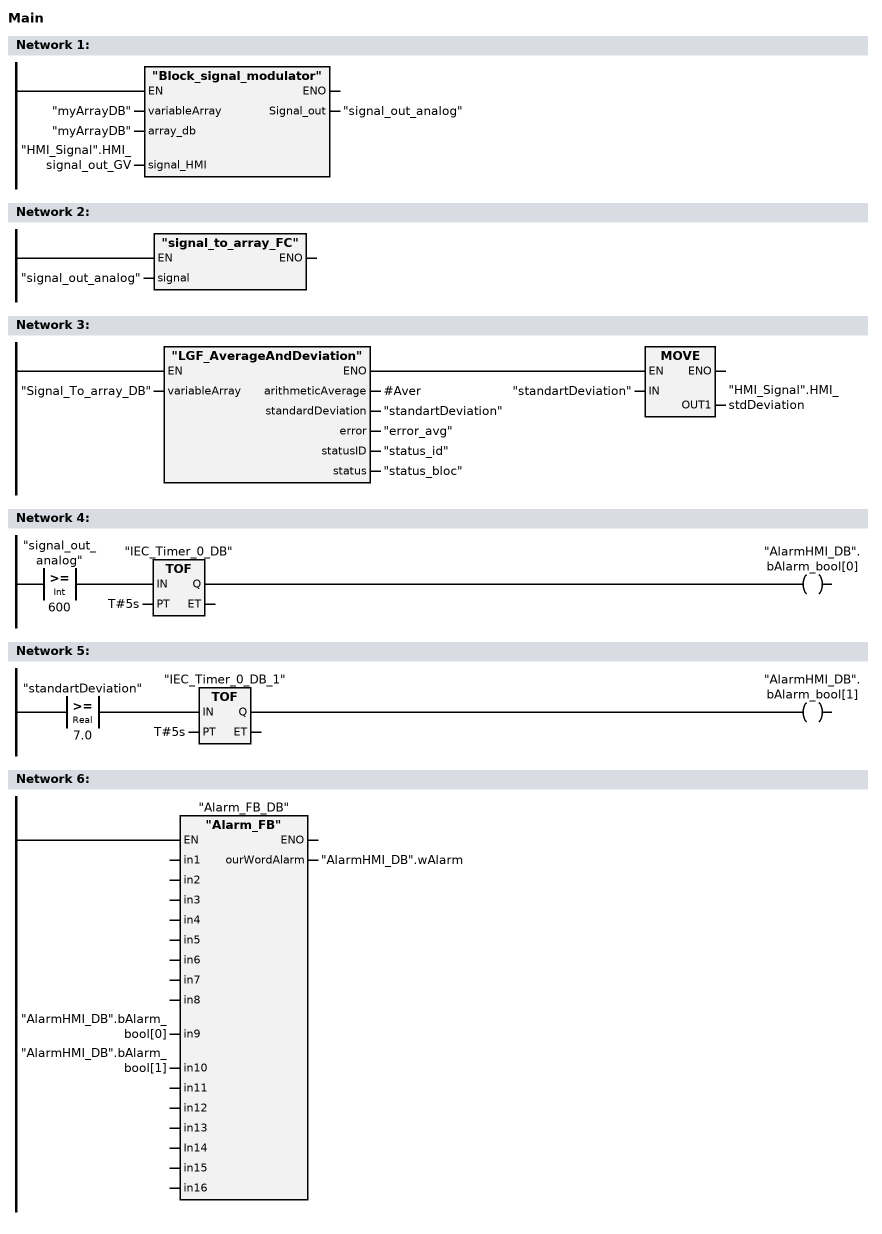
   RUNG wire#powerrail
      "Block_signal_modulator"(variableArray := "myArrayDB", array_db := "myArrayDB", signal_HMI := "HMI_Signal".HMI_signal_out_GV, Signal_out => "signal_out_analog")
   END_RUNG
   // the same network as SCL:
   "Block_signal_modulator"(variableArray := "myArrayDB",
                           array_db := "myArrayDB",
                           signal_HMI := "HMI_Signal".HMI_signal_out_GV,
                           Signal_out => "signal_out_analog");
END_REGION

REGION Network 2
   RUNG wire#powerrail
      "signal_to_array_FC"(signal := "signal_out_analog")
   END_RUNG
   // the same network as SCL:
   "signal_to_array_FC"(signal := "signal_out_analog");
END_REGION

REGION Network 3
   RUNG wire#powerrail
      "LGF_AverageAndDeviation"(variableArray := "Signal_To_array_DB", arithmeticAverage => #Aver, standardDeviation => "standartDeviation", error => "error_avg", statusID => "status_id", status => "status_bloc")
      Move(in := "standartDeviation", out1 => "HMI_Signal".HMI_stdDeviation)
   END_RUNG
   // the same network as SCL:
   "LGF_AverageAndDeviation"(variableArray := "Signal_To_array_DB",
                           arithmeticAverage => #Aver,
                           standardDeviation => "standartDeviation",
                           error => "error_avg",
                           statusID => "status_id",
                           status => "status_bloc",
                           ENO => #_w1);
   IF #_w1 THEN "HMI_Signal".HMI_stdDeviation := "standartDeviation"; END_IF;
END_REGION

REGION Network 4
   "IEC_Timer_0_DB".TOF(IN := "signal_out_analog" >= 600, PT := T#5s);
   "AlarmHMI_DB".bAlarm_bool[0] := "IEC_Timer_0_DB".Q;
END_REGION

REGION Network 5
   "IEC_Timer_0_DB_1".TOF(IN := "standartDeviation" >= 7.0, PT := T#5s);
   "AlarmHMI_DB".bAlarm_bool[1] := "IEC_Timer_0_DB_1".Q;
END_REGION

REGION Network 6
   RUNG wire#powerrail
      "Alarm_FB_DB"(in1 :=, in2 :=, in3 :=, in4 :=, in5 :=, in6 :=, in7 :=, in8 :=, in9 := "AlarmHMI_DB".bAlarm_bool[0], in10 := "AlarmHMI_DB".bAlarm_bool[1], in11 :=, in12 :=, in13 :=, In14 :=, in15 :=, in16 :=, ourWordAlarm => "AlarmHMI_DB".wAlarm)
   END_RUNG
   // the same network as SCL:
   "Alarm_FB_DB"(in9 := "AlarmHMI_DB".bAlarm_bool[0],   // "Alarm_FB"
                 in10 := "AlarmHMI_DB".bAlarm_bool[1],
                 ourWordAlarm => "AlarmHMI_DB".wAlarm);
END_REGION
END_ORGANIZATION_BLOCK

// folder: 4 Math operations

FUNCTION "LGF_AverageAndDeviation" : Void   // FC10006, SCL
{ S7_Optimized_Access := 'TRUE' }
   VAR_INPUT
      variableArray : Variant;
   END_VAR
   VAR_OUTPUT
      arithmeticAverage : Real;
      standardDeviation : Real;
      error : Bool;
      statusID : UInt;
      status : Word;
   END_VAR
   VAR_TEMP
      tempArraySize : UDInt;
      tempSizeCounter : Int;
      tempInternalError : Int;
      tempActValueInt : Int;
      tempActValueUInt : UInt;
      tempActValueDInt : DInt;
      tempActValueUDInt : UDInt;
      tempActValueUSInt : USInt;
      tempActValueSInt : SInt;
      tempActValueReal : Real;
      tempArithmeticAverage : Real;
      tempStandardDeviation : Real;
   END_VAR
   VAR CONSTANT
      NO_ERROR : Word := 16#0000;
      NO_CURRENT_JOBS : Word := 16#7000;
      NO_ARRAY : Word := 16#8200;
      WRONG_TYPE : Word := 16#8201;
      ERROR_IN_THIS_BLOCK : UInt := 1;
      ERROR_MOVE_BLK_VARIANT : UInt := 2;
   END_VAR
BEGIN
   //=============================================================================
   // SIEMENS AG
   // (c)Copyright 2017
   //-----------------------------------------------------------------------------
   // Library:       LGF (Library General Functions)
   // Tested with:   CPU1212C DC/DC/DC FW:V4.2
   // Engineering:   TIA Portal V14 Update 1
   // Restrictions:  -
   // Requirements:  PLC (S7-1200 / S7-1500)
   // Functionality: This function calculates the arithmetic average and the
   //                standard Deviation of a array of numbers
   //-----------------------------------------------------------------------------
   // Change log table:
   // Version  Date        In charge / Changes applied
   // 01.00.00 19.08.2015  Siemens Industry Online Support
   //                      First released version
   // 01.00.01 16.11.2015  Siemens Industry Online Support
   //                      Bug fix at WRONG_TYPE:  #error := true
   // 01.00.02 02.01.2017  Siemens Industry Online Support
   //                      Upgrade: TIA Portal V14 Update 1
   //=============================================================================

   //set "No current job" status
   #error := false;
   #statusID := #ERROR_IN_THIS_BLOCK;
   #status := #NO_CURRENT_JOBS;

   // Check if the variant-variable is an array if yes cout the elements of the array
   IF NOT (IS_ARRAY(#variableArray)) THEN
     #error := true;
     #statusID := #ERROR_IN_THIS_BLOCK;
     #status := #NO_ARRAY;
     RETURN;
   ELSE
     #tempArraySize := CountOfElements(#variableArray);
   END_IF;

   CASE TypeOfElements(#variableArray) OF
     Int:
       // Calculation of the arithmetic average
       #tempArithmeticAverage := 0;
       FOR #tempSizeCounter := 0 TO UDINT_TO_INT(#tempArraySize) - 1 DO
         #tempInternalError := MOVE_BLK_VARIANT(SRC := #variableArray,
                                                COUNT := 1,
                                                SRC_INDEX := #tempSizeCounter,
                                                DEST_INDEX := 0,
                                                DEST => #tempActValueInt);

         #tempArithmeticAverage := #tempArithmeticAverage + INT_TO_REAL(#tempActValueInt);
       END_FOR;

       #tempArithmeticAverage := #tempArithmeticAverage / UDINT_TO_REAL(#tempArraySize);

       //------------------------------------------
       //Calculation of the standardDeviation
       #tempStandardDeviation := 0;
       FOR #tempSizeCounter := 0 TO UDINT_TO_INT(#tempArraySize) - 1 DO
         #tempInternalError := MOVE_BLK_VARIANT(SRC := #variableArray,
                                                COUNT := 1,
                                                SRC_INDEX := #tempSizeCounter,
                                                DEST_INDEX := 0,
                                                DEST => #tempActValueInt);

         #tempStandardDeviation := #tempStandardDeviation + SQR((INT_TO_REAL(#tempActValueInt) - #tempArithmeticAverage));
       END_FOR;

       #tempStandardDeviation := #tempStandardDeviation / UDINT_TO_REAL(#tempArraySize);
       #tempStandardDeviation := SQRT(#tempStandardDeviation);

       //-------------------------------------------
     DInt:
       // Calculation of the arithmetic average
       #tempArithmeticAverage := 0;
       FOR #tempSizeCounter := 0 TO UDINT_TO_INT(#tempArraySize) - 1 DO
         #tempInternalError := MOVE_BLK_VARIANT(SRC := #variableArray,
                                                COUNT := 1,
                                                SRC_INDEX := #tempSizeCounter,
                                                DEST_INDEX := 0,
                                                DEST => #tempActValueDInt);

         #tempArithmeticAverage := #tempArithmeticAverage + DINT_TO_REAL(#tempActValueDInt);
       END_FOR;

       #tempArithmeticAverage := #tempArithmeticAverage / UDINT_TO_REAL(#tempArraySize);

       //------------------------------------------
       //Calculation of the standardDeviation
       #tempStandardDeviation := 0;
       FOR #tempSizeCounter := 0 TO UDINT_TO_INT(#tempArraySize) - 1 DO
         #tempInternalError := MOVE_BLK_VARIANT(SRC := #variableArray,
                                                COUNT := 1,
                                                SRC_INDEX := #tempSizeCounter,
                                                DEST_INDEX := 0,
                                                DEST => #tempActValueDInt);

         #tempStandardDeviation := #tempStandardDeviation + SQR((DINT_TO_REAL(#tempActValueDInt) - #tempArithmeticAverage));
       END_FOR;

       #tempStandardDeviation := #tempStandardDeviation / UDINT_TO_REAL(#tempArraySize);
       #tempStandardDeviation := SQRT(#tempStandardDeviation);

       //-------------------------------------------
     UInt:
       // Calculation of the arithmetic average
       #tempArithmeticAverage := 0;
       FOR #tempSizeCounter := 0 TO UDINT_TO_INT(#tempArraySize) - 1 DO
         #tempInternalError := MOVE_BLK_VARIANT(SRC := #variableArray,
                                                COUNT := 1,
                                                SRC_INDEX := #tempSizeCounter,
                                                DEST_INDEX := 0,
                                                DEST => #tempActValueUInt);

         #tempArithmeticAverage := #tempArithmeticAverage + UINT_TO_REAL(#tempActValueUInt);
       END_FOR;

       #tempArithmeticAverage := #tempArithmeticAverage / UDINT_TO_REAL(#tempArraySize);

       //------------------------------------------
       //Calculation of the standardDeviation
       #tempStandardDeviation := 0;
       FOR #tempSizeCounter := 0 TO UDINT_TO_INT(#tempArraySize) - 1 DO
         #tempInternalError := MOVE_BLK_VARIANT(SRC := #variableArray,
                                                COUNT := 1,
                                                SRC_INDEX := #tempSizeCounter,
                                                DEST_INDEX := 0,
                                                DEST => #tempActValueUInt);

         #tempStandardDeviation := #tempStandardDeviation + SQR((UINT_TO_REAL(#tempActValueUInt) - #tempArithmeticAverage));
       END_FOR;

       #tempStandardDeviation := #tempStandardDeviation / UDINT_TO_REAL(#tempArraySize);
       #tempStandardDeviation := SQRT(#tempStandardDeviation);

       //-------------------------------------------
     UDInt:
       // Calculation of the arithmetic average
       #tempArithmeticAverage := 0;
       FOR #tempSizeCounter := 0 TO UDINT_TO_INT(#tempArraySize) - 1 DO
         #tempInternalError := MOVE_BLK_VARIANT(SRC := #variableArray,
                                                COUNT := 1,
                                                SRC_INDEX := #tempSizeCounter,
                                                DEST_INDEX := 0,
                                                DEST => #tempActValueUDInt);

         #tempArithmeticAverage := #tempArithmeticAverage + UDINT_TO_REAL(#tempActValueUDInt);
       END_FOR;

       #tempArithmeticAverage := #tempArithmeticAverage / UDINT_TO_REAL(#tempArraySize);

       //------------------------------------------
       //Calculation of the standardDeviation
       #tempStandardDeviation := 0;
       FOR #tempSizeCounter := 0 TO UDINT_TO_INT(#tempArraySize) - 1 DO
         #tempInternalError := MOVE_BLK_VARIANT(SRC := #variableArray,
                                                COUNT := 1,
                                                SRC_INDEX := #tempSizeCounter,
                                                DEST_INDEX := 0,
                                                DEST => #tempActValueUDInt);

         #tempStandardDeviation := #tempStandardDeviation + SQR((UDINT_TO_REAL(#tempActValueUDInt) - #tempArithmeticAverage));
       END_FOR;

       #tempStandardDeviation := #tempStandardDeviation / UDINT_TO_REAL(#tempArraySize);
       #tempStandardDeviation := SQRT(#tempStandardDeviation);

       //-------------------------------------------;
     USInt:
       // Calculation of the arithmetic average
       #tempArithmeticAverage := 0;
       FOR #tempSizeCounter := 0 TO UDINT_TO_INT(#tempArraySize) - 1 DO
         #tempInternalError := MOVE_BLK_VARIANT(SRC := #variableArray,
                                                COUNT := 1,
                                                SRC_INDEX := #tempSizeCounter,
                                                DEST_INDEX := 0,
                                                DEST => #tempActValueUSInt);

         #tempArithmeticAverage := #tempArithmeticAverage + USINT_TO_REAL(#tempActValueUSInt);
       END_FOR;

       #tempArithmeticAverage := #tempArithmeticAverage/ UDINT_TO_REAL(#tempArraySize);

       //------------------------------------------
       //Calculation of the standardDeviation
       #tempStandardDeviation := 0;
       FOR #tempSizeCounter := 0 TO UDINT_TO_INT(#tempArraySize) - 1 DO
         #tempInternalError := MOVE_BLK_VARIANT(SRC := #variableArray,
                                                COUNT := 1,
                                                SRC_INDEX := #tempSizeCounter,
                                                DEST_INDEX := 0,
                                                DEST => #tempActValueUSInt);

         #tempStandardDeviation := #tempStandardDeviation + SQR((USINT_TO_REAL(#tempActValueUSInt) - #tempArithmeticAverage));
       END_FOR;

       #tempStandardDeviation := #tempStandardDeviation / UDINT_TO_REAL(#tempArraySize);
       #tempStandardDeviation := SQRT(#tempStandardDeviation);

       //-------------------------------------------
     SInt:
       // Calculation of the arithmetic average
       #tempArithmeticAverage := 0;
       FOR #tempSizeCounter := 0 TO UDINT_TO_INT(#tempArraySize) - 1 DO
         #tempInternalError := MOVE_BLK_VARIANT(SRC := #variableArray,
                                                COUNT := 1,
                                                SRC_INDEX := #tempSizeCounter,
                                                DEST_INDEX := 0,
                                                DEST => #tempActValueSInt);

         #tempArithmeticAverage := #tempArithmeticAverage + SINT_TO_REAL(#tempActValueSInt);
       END_FOR;

       #tempArithmeticAverage := #tempArithmeticAverage / UDINT_TO_REAL(#tempArraySize);

       //------------------------------------------
       //Calculation of the standardDeviation
       #tempStandardDeviation := 0;
       FOR #tempSizeCounter := 0 TO UDINT_TO_INT(#tempArraySize) - 1 DO
         #tempInternalError := MOVE_BLK_VARIANT(SRC := #variableArray,
                                                COUNT := 1,
                                                SRC_INDEX := #tempSizeCounter,
                                                DEST_INDEX := 0,
                                                DEST => #tempActValueSInt);

         #tempStandardDeviation := #tempStandardDeviation + SQR((SINT_TO_REAL(#tempActValueSInt) - #tempArithmeticAverage));
       END_FOR;

       #tempStandardDeviation := #tempStandardDeviation / UDINT_TO_REAL(#tempArraySize);
       #tempStandardDeviation := SQRT(#tempStandardDeviation);

       //-------------------------------------------
     Real:
       // Calculation of the arithmetic average
       #tempArithmeticAverage := 0;
       FOR #tempSizeCounter := 0 TO UDINT_TO_INT(#tempArraySize) - 1 DO
         #tempInternalError := MOVE_BLK_VARIANT(SRC := #variableArray,
                                                COUNT := 1,
                                                SRC_INDEX := #tempSizeCounter,
                                                DEST_INDEX := 0,
                                                DEST => #tempActValueReal);

         #tempArithmeticAverage := #tempArithmeticAverage + #tempActValueReal;
       END_FOR;

       #tempArithmeticAverage := #tempArithmeticAverage / UDINT_TO_REAL(#tempArraySize);

       //------------------------------------------
       //Calculation of the standardDeviation
       #tempStandardDeviation := 0;
       FOR #tempSizeCounter := 0 TO UDINT_TO_INT(#tempArraySize) - 1 DO
         #tempInternalError := MOVE_BLK_VARIANT(SRC := #variableArray,
                                                COUNT := 1,
                                                SRC_INDEX := #tempSizeCounter,
                                                DEST_INDEX := 0,
                                                DEST => #tempActValueReal);

         #tempStandardDeviation := #tempStandardDeviation + SQR((#tempActValueReal - #tempArithmeticAverage));
       END_FOR;

       #tempStandardDeviation := #tempStandardDeviation / UDINT_TO_REAL(#tempArraySize);
       #tempStandardDeviation := SQRT(#tempStandardDeviation);

       //-------------------------------------------
     ELSE
       #error := true;
       #statusID := #ERROR_IN_THIS_BLOCK;
       #status := #WRONG_TYPE;
       RETURN;
   END_CASE;
   #arithmeticAverage := #tempArithmeticAverage;
   #standardDeviation := #tempStandardDeviation;

   IF #tempInternalError > 1 THEN
     #error := true;
     #statusID := #ERROR_MOVE_BLK_VARIANT;
     #status := INT_TO_WORD(#tempInternalError);
     RETURN;
   END_IF;

   #status := #NO_ERROR;
END_FUNCTION

// folder: 7 Signal generators

FUNCTION_BLOCK "LGF_Frequency"   // FB10024, SCL
{ S7_Optimized_Access := 'TRUE' }
   VAR_INPUT
      frequency : Real;   // Input in Hz
      pulsePauseRatio : Real := 1.0;   // Pulse pause ratio
   END_VAR
   VAR_OUTPUT
      clock : Bool;   // -
      countdown : Time;   // -
   END_VAR
   VAR
      instTofTimePulse : TOF_TIME;   // -
      instTofTimePause : TOF_TIME;   // -
      statFrequency : Real;   // -
      statTimePeriod : Time;   // -
      statTimePulse : Time;   // -
      statTimePause : Time;   // -
      statPulsePauseRatio : Real;   // -
   END_VAR
   VAR_TEMP
      tempPulseRate : Real;   // -
      tempPauseRate : Real;   // -
   END_VAR
   VAR CONSTANT
      NULL : Real := 0.0;   // -
   END_VAR
BEGIN
   //=============================================================================
   // SIEMENS AG
   // (c)Copyright 2017
   //-----------------------------------------------------------------------------
   // Library:       LGF (Library General Functions)
   // Tested with:   CPU1214C DC/DC/DC FW:V4.2
   // Engineering:   TIA Portal V14
   // Restrictions:  -
   // Requirements:  PLC (S7-1200, S7-1500)
   // Functionality: Generates frequency signal
   //-----------------------------------------------------------------------------
   // Change log table:
   // Version  Date        Expert in charge / Changes applied
   // 01.00.00 19.08.2015  Siemens Industry Online Support
   //                      First released version
   // 01.01.00 25.05.2016  Siemens Industry Online Support
   //                      New function: pulse pause ratio
   // 01.01.01 26.05.2016  Siemens Industry Online Support
   //                      Add comments
   // 01.01.02 02.01.2017  Siemens Industry Online Support
   //                      Upgrade: TIA Portal V14 Update 1
   //=============================================================================

   IF (#frequency <= #NULL) OR (#pulsePauseRatio <= #NULL)  // If input is <= 0.0 : block is off
   THEN
     #clock := FALSE;
     #countdown := t#0s;
   ELSE
     // assign frequency and pulse pause ratio one time 
     IF #statFrequency <> #frequency OR #statPulsePauseRatio <> #pulsePauseRatio THEN
       RESET_TIMER(TIMER := #instTofTimePause);
       RESET_TIMER(TIMER := #instTofTimePulse);

       #tempPulseRate := #pulsePauseRatio / (#pulsePauseRatio + 1); // Calculate pulse rate   
       #tempPauseRate := 1.0 - #tempPulseRate;                      // Calculate pause rate   
       #statTimePeriod := T_CONV(REAL_TO_UDINT((1000.0 / #frequency)));                 // Calculate period time 
       #statTimePulse := T_CONV(REAL_TO_UDINT((1000.0 * #tempPulseRate / #frequency))); // Calculate pulse time   
       #statTimePause := T_CONV(REAL_TO_UDINT((1000.0 * #tempPauseRate / #frequency))); // Calculate pause time
       #statFrequency := #frequency;
       #statPulsePauseRatio := #pulsePauseRatio;
     END_IF;

     // TOF_off expired >> Start again
     #instTofTimePulse(IN := NOT #instTofTimePause.Q,
                       PT := #statTimePulse);
     #countdown := #statTimePulse - #instTofTimePulse.ET;

     #instTofTimePause(IN := #instTofTimePulse.Q,
                       PT := #statTimePause);

     IF #countdown = t#0s THEN
       #countdown := #statTimePause - #instTofTimePause.ET;
     END_IF;

     #clock := #instTofTimePulse.Q; // Assign ouptut 
   END_IF;
END_FUNCTION_BLOCK

// folder: 8 Technology operations

FUNCTION_BLOCK "LGF_LimRateOfChangeAdvanced"   // FB10033, SCL
{ S7_Optimized_Access := 'TRUE' }
VERSION : 0.1
   VAR_INPUT
      inputValue : Real;   // input value
      setPosUpRateLim : Real;   // limit up rate of change in positiv range (1/second)
      setPosDownRateLim : Real;   // limit down rate of change in positiv range (1/second)
      setNegUpRateLim : Real;   // limit up rate of change in nagativ range (1/second)
      setNegDownRateLim : Real;   // limit down rate of change in nagativ range (1/second)
      setHighLim : Real;   // high limit
      setLowLim : Real;   // low limit
      processValue : Real;   // process value
      defaultOutValue : Real;   // default output value
      onDefaultOutValue : Bool;   // default output value on (outputValue=defaultOutValue)
      track : Bool;   // tracking (outVal=inputValue)
      manOp : Bool;   // manual mode on (outputValue=processValue)
      reset : Bool;   // complete restart
      callOB : OB_Cyclic;   // cyclic interrupt OB
   END_VAR
   VAR_OUTPUT
      outputValue : Real;   // output value
      posUpRateLim : Bool;   // up rate limit in positiv range reached
      posDownRateLim : Bool;   // down rate limit in positiv range reached
      negUpRateLim : Bool;   // up rate limit in negative range reached
      negDownRateLim : Bool;   // down rate limit in negativ range reached
      highLim : Bool;   // high limit reached
      lowLim : Bool;   // low limit reached
      error : Bool;   // "0" = no error; "1" = error
      statusID : UInt;   // Error destination: "1" = LGFLimRateOfChangeAdvanced; "2" = QRY_CINT
      status : Word;   // status and error codes
   END_VAR
   VAR
      statPrevOutputValue : Real := 0.0;   // -
      statManOp : Bool;   // -
   END_VAR
   VAR_TEMP
      tempPosUp : Bool;   // -
      tempPosDown : Bool;   // -
      tempNegUp : Bool;   // -
      tempNegDown : Bool;   // -
      tempHighLim : Bool;   // -
      tempLowLim : Bool;   // -
      tempCycleReal : Real;   // -
      tempOutv : Real;   // -
      tempVar : Real;   // -
      tempCycleTime : UDInt;   // -
      tempCyclePhase : UDInt;   // -
      tempCycleStatus : Word;   // -
      tempReadTimeStatus : Int;   // -
   END_VAR
   VAR CONSTANT
      NO_ERROR : Word := 16#0000;   // -
      OB_UNAVAILABLE : Word := 16#8200;   // -
      HIGHLIM_UNDER_LOWLIM : Word := 16#8201;   // -
      NEG_RATE_OF_CHANGE : Word := 16#8202;   // -
      ERROR_IN_THIS_BLOCK : UInt := 1;   // -
      ERROR_QRY_CINT : UInt := 2;   // -
   END_VAR
BEGIN
   //=============================================================================
   // Siemens AG
   // (c)Copyright 2017
   //-----------------------------------------------------------------------------
   // Library:       LGF(Library General Functions)
   // Tested with:   CPU1212C DC/DC/DC FW:V4.2
   // Engineering:   TIA Portal V14 Update 1
   // Restrictions:  only callable just in cyclic interrupt OB
   // Requirements:  PLC (S7-1200 / S7-1500)
   // Functionality: This function block generates a ramp function from a step 
   //                function with advanced modes and settings.  
   //-----------------------------------------------------------------------------
   // Change log table:
   // Version  Date        In charge / Changes applied
   // 01.00.00 21.06.2016  Siemens Industry Online Support
   //                      First released version
   // 01.00.01 02.01.2017  Siemens Industry Online Support
   //                      Upgrade: TIA Portal V14 Update 1
   //-----------------------------------------------------------------------------
   //Status Codes:
   // 16#0000:  No errors
   // 16#8200:  Call OB unavailable
   // 16#8201:  Paramater for high limit lower thal low limit
   // 16#8202:  Negativ value for the rate of change parameter
   //=============================================================================

   // Initialize
   #error := FALSE;
   #statusID := #ERROR_IN_THIS_BLOCK;
   #status := #NO_ERROR;

   //***// get sample time, according to the cyclic interrupt OB number
   #tempReadTimeStatus := QRY_CINT(OB_NR := #callOB, CYCLE => #tempCycleTime,
                                   PHASE => #tempCyclePhase, STATUS => #tempCycleStatus);
   #tempCycleReal := UDINT_TO_REAL(#tempCycleTime) / 1.0e6; // Time in seconds

   // Generate error message of the QRY_CINT function
   IF (#tempReadTimeStatus <> 0) THEN
     #error := TRUE;
     #statusID := #ERROR_QRY_CINT;
     #status := INT_TO_WORD(#tempReadTimeStatus);
     RETURN;
   END_IF;

   // Generate error message when OB unavailable
   IF #tempCycleStatus = 16#0000 THEN
     #error := TRUE;
     #statusID := #ERROR_IN_THIS_BLOCK;
     #status := #OB_UNAVAILABLE;
     RETURN;
   END_IF;

   IF #setHighLim < #setLowLim THEN
     #error := TRUE;
     #statusID := #ERROR_IN_THIS_BLOCK;
     #status := #HIGHLIM_UNDER_LOWLIM;
     RETURN;
   END_IF;

   IF (#setNegDownRateLim < 0.0) OR (#setNegUpRateLim < 0.0)
     OR (#setPosDownRateLim < 0.0) OR (#setPosUpRateLim < 0.0)
   THEN
     #error := TRUE;
     #statusID := #ERROR_IN_THIS_BLOCK;
     #status := #NEG_RATE_OF_CHANGE;
     RETURN;
   END_IF;

   // Initialize temp variable
   #tempPosUp := FALSE;
   #tempPosDown := FALSE;
   #tempNegUp := FALSE;
   #tempNegDown := FALSE;
   #tempHighLim := FALSE;
   #tempLowLim := FALSE;
   #tempOutv := #inputValue;

   // RESTART
   IF #reset
   THEN
     #statManOp := FALSE;    // reset manual mode flag 
     IF #onDefaultOutValue
       // preset output
     THEN
       #tempOutv := #defaultOutValue;
       // limitation of output
       IF #tempOutv >= #setHighLim
       THEN
         // High limitation
         #tempOutv := #setHighLim;
         #tempHighLim := TRUE;
       END_IF;

       IF #tempOutv <= #setLowLim
       THEN
         // Low limitation
         #tempOutv := #setLowLim;
         #tempLowLim := TRUE;
       END_IF;
     ELSE
       // reset output
       #tempOutv := 0.0;
     END_IF;
   ELSE

     // OPERATING MODES
     // -------------------------------------------------------
     IF #manOp
     THEN
       //---// MANUAL MODE
       // bumples switch between manual mode and auto mode    
       #tempOutv := #processValue;
       // Keep manual mode until setpoint in the space of low and high limit
       #statManOp := TRUE;
     ELSE
       //---// AUTOMATIC MODE
       IF #onDefaultOutValue
       THEN
         // preset output by default value
         #tempOutv := #defaultOutValue;
       ELSE
         IF #track
         THEN
           // output has same value as input
           #tempOutv := #inputValue;
         ELSE
           // REGULAR FUNCTION                    
           // Negativ range
           IF #statPrevOutputValue < 0
           THEN
             IF #statPrevOutputValue > #inputValue
             THEN
               // limited rate of change
               #tempVar := #statPrevOutputValue - #setNegUpRateLim * #tempCycleReal;
               IF #inputValue < #tempVar
               THEN
                 // Setpoint not reached yet
                 // set notification for up rate limit in neg range              
                 #tempNegUp := TRUE;
                 #tempOutv := #tempVar;
               END_IF;
             ELSE
               IF #setNegDownRateLim = 0.0
               THEN
                 // set notification for down rate limit in neg range              
                 #tempNegDown := TRUE;
                 IF #inputValue <= 0.0
                 THEN
                   #tempOutv := #inputValue;
                 ELSE
                   #tempOutv := 0.0;
                 END_IF;
               ELSE
                 IF #inputValue <= 0.0
                 THEN
                   // limited rate of change
                   #tempVar := #statPrevOutputValue + #setNegDownRateLim * #tempCycleReal;
                   IF #inputValue > #tempVar
                   THEN
                     // set notification for down rate limit in neg range
                     #tempNegDown := TRUE;
                     #tempOutv := #tempVar;
                   END_IF;
                 ELSE
                   // changeover between neg. and pos. range
                   // period till zero-crossing
                   #tempVar := - #statPrevOutputValue / #setNegDownRateLim;

                   IF #tempVar <= #tempCycleReal
                   THEN
                     // period till zero-crossing shorten than sample time
                     // limited rate of change
                     #tempVar := (#tempCycleReal - #tempVar) * #setPosUpRateLim;

                     IF #inputValue > #tempVar
                     THEN
                       // set notification for rate limit 
                       #tempNegDown := FALSE;
                       #tempPosUp := TRUE;
                       #tempOutv := #tempVar;
                     END_IF;
                   ELSE
                     // set notification for rate limit
                     #tempNegDown := TRUE;
                     #tempPosUp := FALSE;
                     #tempOutv := #statPrevOutputValue + #tempCycleReal * #setNegDownRateLim;
                   END_IF;
                 END_IF;
               END_IF;
             END_IF;
           ELSE
             // Positiv range + 0                        
             IF #statPrevOutputValue < #inputValue
             THEN
               // limited rate of change
               #tempVar := #statPrevOutputValue + #setPosUpRateLim * #tempCycleReal;
               IF #inputValue > #tempVar
               THEN
                 // set notification for up rate limit in pos range              
                 #tempPosUp := TRUE;
                 #tempOutv := #tempVar;
               END_IF;
             END_IF;

             IF #statPrevOutputValue >= #inputValue
             THEN
               IF #setPosDownRateLim = 0.0
               THEN
                 // set notification for down rate limit in pos range              
                 #tempPosDown := TRUE;
                 IF #inputValue >= 0.0
                 THEN
                   #tempOutv := #inputValue;
                 ELSE
                   #tempOutv := 0.0;
                 END_IF;
               ELSE
                 IF #inputValue >= 0.0
                 THEN
                   // limited rate of change
                   #tempVar := #statPrevOutputValue - #setPosDownRateLim * #tempCycleReal;
                   IF #inputValue < #tempVar
                   THEN
                     // set notification for up rate limit in pos range                  
                     #tempPosDown := TRUE;
                     #tempOutv := #tempVar;
                   END_IF;
                 ELSE  // changeover between pos. and neg. range
                   // period till zero-crossing
                   #tempVar := #statPrevOutputValue / #setPosDownRateLim;

                   IF #tempVar <= #tempCycleReal
                   THEN
                     // limited rate of change
                     #tempVar := - (#tempCycleReal - #tempVar) * #setNegUpRateLim;

                     IF #inputValue < #tempVar
                     THEN
                       // set notification for rate limit
                       #tempPosDown := False;
                       #tempNegUp := TRUE;
                       #tempOutv := #tempVar;
                     END_IF;
                   ELSE
                     // set notification for rate limit
                     #tempPosDown := TRUE;
                     #tempNegUp := FALSE;
                     #tempOutv := #statPrevOutputValue - #tempCycleReal * #setPosDownRateLim;
                   END_IF;
                 END_IF;
               END_IF;
             END_IF;
           END_IF;
         END_IF;
       END_IF;

       // high/low level limitation
       IF #tempOutv >= #setHighLim
       THEN
         #tempHighLim := TRUE;
         IF NOT #statManOp
         THEN
           #tempOutv := #setHighLim;
           // correct up rate limit notification                
           IF #tempOutv - #statPrevOutputValue < #setPosUpRateLim * #tempCycleReal
           THEN
             #tempPosUp := FALSE;
           END_IF;
         END_IF;
       ELSE
         IF #tempOutv <= #setLowLim
         THEN
           #tempLowLim := TRUE;
           IF NOT #statManOp
           THEN
             #tempOutv := #setLowLim;
             // correct up rate limit notification  
             IF #statPrevOutputValue - #tempOutv < #setNegUpRateLim * #tempCycleReal
             THEN
               #tempNegUp := FALSE;
             END_IF;
           END_IF;
         ELSE
           // reset manual mode flag when tempOutv between upper and lower limit        
           #statManOp := FALSE;
         END_IF;
       END_IF;
     END_IF;
   END_IF;


   // update output parameters
   #outputValue := #tempOutv;    // output
   #statPrevOutputValue := #tempOutv;
   #posUpRateLim := #tempPosUp;
   #posDownRateLim := #tempPosDown;
   #negUpRateLim := #tempNegUp;
   #negDownRateLim := #tempNegDown;
   #highLim := #tempHighLim;
   #lowLim := #tempLowLim;
END_FUNCTION_BLOCK

(* ===== HMI "HMI_RT_1" =====
system functions are stored by id; their names below are inferred from use
connection "HMI_Connection_1": ETHERNET, SMART_S7_1500_OMS

HMI tags "Default tag table"
   "Tag_ScreenNumber" : UInt, internal
   "signal_out_analog" : Int = PLC signal_out_analog AT %MW32, 1 s
   "standartDeviation" : Real = PLC standartDeviation AT %MD34, 1 s

HMI tags "HMI_signal"
   "HMI_Signal_HMI_signal_out_GV" : Int = PLC HMI_Signal.HMI_signal_out_GV, 1 s
   "HMI_Signal_HMI_stdDeviation" : Real = PLC HMI_Signal.HMI_stdDeviation, 1 s

HMI tags "Alarm_HMI"
   "AlarmHMI_DB_wAlarm" : Word = PLC AlarmHMI_DB.wAlarm, 1 s

discrete alarms
   1: 'Ошибка 1', class Errors, trigger "AlarmHMI_DB_wAlarm" bit 0
   2: 'Ошибка 2', class Errors, trigger "AlarmHMI_DB_wAlarm" bit 1
   3: 'Ошибка 3', class Errors, trigger "AlarmHMI_DB_wAlarm" bit 2

Template "Template_1" 800x480
   Button "Template_Button" at 722,440 size 55x39; TextOff 'Text'
   Button "Template_Button_1" at 622,440 size 55x39; TextOff 'Text'
   Button "Template_Button_2" at 522,440 size 55x39; TextOff 'Text'
   Button "Template_Button_3" at 422,440 size 55x39; TextOff 'Text'
   Button "Template_Button_4" at 322,440 size 55x39; TextOff 'Text'
   Button "Template_Button_5" at 222,440 size 55x39; TextOff 'Text'
   Button "Alarms" at 122,440 size 55x39; TextOff 'Alarms'; PictureOff "AlarmDisplay_KTP900_Basic_PN_TR"; PictureOn "AlarmDisplay_KTP900_Basic_PN_TR"
      on Release: function_ef3f5d25("Alarm window_Unacknowledged", -1)
   Button "Template_Button_6" at 22,440 size 55x39; TextOff 'Text'
   SymbolicIOField "Symbolic_IO_Field_Screen" at 2,7 size 691x26; TextOff '0'; TextOn '1'; TextList "TextList_ScreenNames"
      ProcessValue <- "Tag_ScreenNumber"
      on Change: ActivateScreenByNumber("Tag_ScreenNumber", 0)
   DateTimeField "HmiScreenItemData" at 695,20 size 105x20
   DateTimeField "HmiScreenItemData_1" at 695,0 size 105x20

screen "Root screen" 800x480, template "Template_1"
   on GenerateScreen: SetTag("Tag_ScreenNumber", 1)
   TrendView "Trend view_1" at 0,0 size 799x349
   AlarmView "Alarm view_1" at 0,349 size 799x97
*)